FUNCTION_BLOCK StateMonitor_Controller
  (* Version 0.1, 2005-12-19, Oscar Ljungkrantz, Chalmers *)
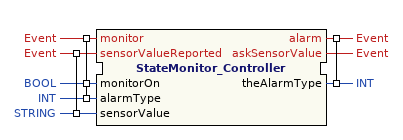
  EVENT_INPUT
    monitor WITH monitorOn, alarmType;
    sensorValueReported WITH sensorValue;
  END_EVENT
  EVENT_OUTPUT
    alarm WITH theAlarmType;
    askSensorValue;
  END_EVENT
  VAR_INPUT
    monitorOn : BOOL;
    alarmType : INT;
    sensorValue : STRING;
  END_VAR
  VAR_OUTPUT
    theAlarmType : INT;
  END_VAR
  VAR
    currentMonitorOn : BOOL := FALSE;
    currentAlarmType : INT := 1;
    currentState : STRING;
  END_VAR
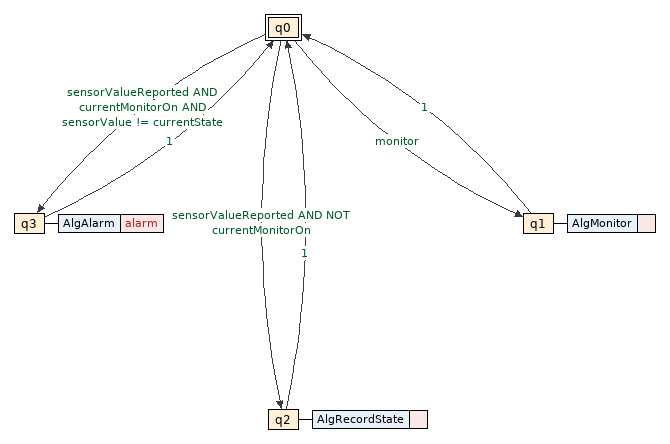
  EC_STATES
    q0;
    q1 : AlgMonitor;
    q2 : AlgRecordState;
    q3 : AlgAlarm -> alarm;
  END_STATES
  EC_TRANSITIONS
    q0 TO q1 := monitor;
    q1 TO q0 := 1;
    q0 TO q2 := sensorValueReported AND NOT currentMonitorOn;
    q2 TO q0 := 1;
    q0 TO q3 := sensorValueReported AND currentMonitorOn AND sensorValue != currentState;
    q3 TO q0 := 1;
  END_TRANSITIONS
  ALGORITHM AlgMonitor IN Java:
		currentMonitorOn = monitorOn;
		currentAlarmType = alarmType;
  END_ALGORITHM
  ALGORITHM AlgRecordState IN Java:
		currentState = sensorValue;
  END_ALGORITHM
  ALGORITHM AlgAlarm IN Java:
		theAlarmType = currentAlarmType;
  END_ALGORITHM
END_FUNCTION_BLOCK
